# B&R Automation Studio project Doctor
Automation Studio 4.9

## Configuration Doctoring

### Cpu.per - 4PPC70_0702_20B/Cpu.per
```iecst
VAR_CONFIG
	AxisKN AT %M0; (* *)
	AxisRPM AT %M70; (* *)
END_VAR
```

## Configuration WndCLTensCtrl

CPU X20CP1586, AutomationRuntime V4.08, Vc V4.15.4

### Task classes (Cpu.sw)
```
DataObjects: Acp10sys
Binaries: vcctext, arialbd, vcmgr, vccshape, vcnet, Visu03, vcdsloc, vcbclass, vcfntttf, vctcal, vcshared, vcrt, vcpkat, Visu01, vccbmp, vcfile, vccbtn, vcalarm, vccnum, vcpdsw, vcdsint, arial, vccovl, vccline, vcpdvnc, vcctrend, vcgclass, vcpfar00, Visu02, vccpopup, vccddbox, vccbar, sysconf, ashwd, asfw, arconfig, Acp10map, acp10cfg, iomap, vccslider, vccdt, vccstr, TCData
Libraries: AsIecCon, astime, NcGlobal, brsystem, sys_lib, Runtime, powerlnk, fileio, Operator, AsBrMath, dataobj, vcresman
```

### PvMap.vvm - X20CP1586/PvMap.vvm
```iecst
(*Simulation model input parameters*)
VAR_CONFIG
	Cyclic#3.::gControl.Winder.Power AT %Q.::SimModel:SimulationModel.Enable; (*Enable simulation modell if machine is ready*)
	Cyclic#3.::gControl.Line.SetVelocity AT %Q.::SimModel:SetLineVelocity; (*Connect control structure with simulation model*)
	Cyclic#3.::gControl.Winder.SetVelocity AT %Q.::SimModel:SetWinderVelocity; (*Connect control structure with simulation model*)
	Cyclic#3.::gControl.Winder.VelocityCorrection AT %Q.::SimModel:WinderVelocityCorrection; (*Connect control structure with simulation model*)
	Cyclic#3.::gControl.Winder.SetMotorTorque AT %Q.::SimModel:SetMotorTorque; (*Connect control structure with simulation model*)
	Cyclic#3.::gControl.Winder.InitSpeedController AT %Q.::SimModel:InitSpeedController; (*Connect control structure with simulation model*)
	Cyclic#3.::gControl.Winder.ActProportionalGain AT %Q.::SimModel:ActProportionalGain; (*Connect control structure with simulation model*)
	Cyclic#3.::gControl.Winder.ActIntegrationTime AT %Q.::SimModel:ActIntegrationTime; (*Connect control structure with simulation model*)
END_VAR
(*Simulation model output parameters*)
VAR_CONFIG
	::SimModel:SimulationModel.ActLinePosition AT %Q.Cyclic#2.::gControl.Line.ActPosition; (*Connect simulation model with control structure*)
	::SimModel:SimulationModel.ActWinderPosition AT %Q.Cyclic#2.::gControl.Winder.ActPosition; (*Connect simulation model with control structure*)
	::SimModel:SimulationModel.ActMaterialTension AT %Q.Cyclic#2.::gControl.ActMaterialTension; (*Connect simulation model with control structure*)
	::SimModel:SimulationModel.ActLineVelocity AT %Q.Cyclic#2.::gControl.Line.ActVelocity; (*Connect simulation model with control structure*)
	::SimModel:SimulationModel.ActWinderVelocity AT %Q.Cyclic#2.::gControl.Winder.ActVelocity; (*Connect simulation model with control structure*)
	::SimModel:SimulationModel.ActMotorTorque AT %Q.Cyclic#2.::gControl.Winder.ActMotorTorque; (*Connect simulation model with control structure*)
END_VAR
```

## Configuration WndDcrCtrl

### Task classes (Cpu.sw)
```
DataObjects: Acp10sys
Binaries: vcctext, arialbd, vcmgr, vccshape, vcnet, Visu03, vcdsloc, vcbclass, vcfntttf, vctcal, vcshared, vcrt, vcpkat, Visu01, vccbmp, vcfile, vccbtn, vcalarm, vccnum, vcpdsw, vcdsint, arial, vccovl, vccline, vcpdvnc, vcctrend, vcgclass, vcpfar00, Visu02, vccpopup, vccddbox, vccbar, sysconf, ashwd, asfw, iomap, arconfig, Acp10map, acp10cfg, vccslider, vccdt, vccstr, TCData
Libraries: AsIecCon, astime, NcGlobal, brsystem, sys_lib, Runtime, powerlnk, fileio, Operator, AsBrMath, dataobj, vcresman
```

## Logical view

Binary libraries used (declarations not repeated): operator, runtime, astime, AsIecCon, brsystem, sys_lib, AsBrMath, LoopConR, LoopCont, Acp10_MC, Acp10man, Acp10par, NcGlobal, Acp10sim, asstring, standard, vclib, visapi, AsEPL


- Library Logical/Libraries/Library (ANSIC) (no source held here)

### Program Logical/HMI (IEC)

#### Variables.var
```iecst
VAR
	CheckCredentials : BOOL;
	ErrorMessage : STRING[80];
	i : INT;
	Init : BOOL;
	InputPassword : STRING[80]; (*Input taken from HMI*)
	InputUsername : STRING[80]; (*Input taken from HMI*)
	CurrentYear : UINT;
	CurrentSecond : USINT;
	CurrentMonth : USINT;
	CurrentMinute : USINT;
	CurrentHour : USINT;
	CurrentDay : USINT;
	NewYear : UINT;
	NewSecond : USINT;
	NewMonth : USINT;
	NewMinute : USINT;
	NewHour : USINT;
	NewDay : USINT;
	DateTimeSet : UINT; (*Confirms if new date/time was set successfully*)
	SetNewDateTime : BOOL; (*Trigger to apply new date/time*)
	RTC_Get : RTCtime_typ; (*Structure to read current date and time*)
	RTC_Set : RTCtime_typ; (*Structure to set current date and time*)
	Status_RTC : UINT;
	temp_var : BOOL;
END_VAR
```

#### Cyclic.st
```iecst
PROGRAM _CYCLIC
	(* Insert code here *)
	IF(Init = 1)THEN
		Init := 0;
	END_IF

	// Time
	// Reads current date/time from PLC's RTC

	RTC_gettime(ADR(RTC_Get));  // Call PLC's built-in RTC function

	// Update outputs for display
	CurrentYear   := RTC_Get.year;
	CurrentMonth  := RTC_Get.month;
	CurrentDay    := RTC_Get.day;
	CurrentHour   := RTC_Get.hour;
	CurrentMinute := RTC_Get.minute;
	CurrentSecond := RTC_Get.second;

	// Set Date and Time when 'Set Date Time' button is pressed
	IF SetNewDateTime THEN
		IF(temp_var = 0)THEN
			Status_RTC	:= 1;
			temp_var	:= 1;
		END_IF

		RTC_Set.year    := NewYear;
		RTC_Set.month   := NewMonth;
		RTC_Set.day     := NewDay;
		RTC_Set.hour    := NewHour;
		RTC_Set.minute  := NewMinute;
		RTC_Set.second  := NewSecond;

		// Call RTC set function
		Status_RTC := RTC_settime(ADR(RTC_Set));  // Returns TRUE if successful

		IF(Status_RTC = 0)THEN
			SetNewDateTime	:= 0;
			temp_var		:= 0;
		END_IF

	END_IF;

	// Login check
	//	FUNCTION FB_CheckCredentials
	// Credential check
	IF (InputUsername = 'Admin' AND InputPassword = '1234') THEN
		LoginSuccessful := TRUE;
		UserAccessLevel := 1;	// Full access
		CheckCredentials := TRUE;
		ErrorMessage := 'Logged in';
	ELSE
		LoginSuccessful := FALSE;
		UserAccessLevel := 0;	// No input access
		CheckCredentials := FALSE;
		ErrorMessage := 'Wrong user name or password';
	END_IF;

	ErrorMessage := '';   	// Clear any previous message
	InputUsername := '';	// Clear InputUsername field
	InputPassword := '';	// Clear InputPassword field

	IF(Alarm_new = 1)THEN
		Statusdp_alarm	:= 0;
	ELSE
		Statusdp_alarm	:= 1;
	END_IF

END_PROGRAM
```

#### Init.st
```iecst
PROGRAM _INIT
		(*Input of Tension Sensor for 4 axes except main drive *)
	AI1[0]	:= 0;	(*Unwinder Loadcell *)
	AI1[1]	:= 0;	(* Infeed Loadcell *)
	AI1[2]	:= 0;	(* Outfeed Loadcell *)
	AI1[3]	:= 0;	(* Winder Load cell *)
	AI1[4]	:= 0;	(* Dummy Load cell for Main Drive *)

	AI2[0]	:= 0;
	AI2[1]	:= 0;
	AI2[2]	:= 0;
	AI2[3]	:= 0; (*This input is configured for MAIN RPM calculation *)

	(* Input for RPM measurement from drive AI for 4 axes except Winder RPM*)
	AI3[0]	:= 0;   (* Unwinder RPM *)
	AI3[1]	:= 0;	(* Infeed RPM *)
	AI3[2]	:= 0;	(* Outfeed RPM *)
	AI3[3]	:= 0;	(* Winder RPM *)
	AI3[4]	:= 0;	(*This input is configured from AI2[3] for MAIN RPM *)

	AO1[0]	:= 0;
	AO1[1]	:= 0;
	AO1[2]	:= 0;
	AO1[3]	:= 0;

	DI1[0]	:= 0;
	DI1[1]	:= 0;
	DI1[2]	:= 0;
	DI1[3]	:= 0;
	DI1[4]	:= 0;
	DI1[5]	:= 0;
	DI1[6]	:= 0;
	DI1[7]	:= 0;
	DI1[8]	:= 0;
	DI1[9]	:= 0;
	DI1[10]	:= 0;
	DI1[11]	:= 0;

	DI2[0]	:= 0;
	DI2[1]	:= 0;
	DI2[2]	:= 0;
	DI2[3]	:= 0;
	DI2[4]	:= 0;
	DI2[5]	:= 0;
	DI2[6]	:= 0;
	DI2[7]	:= 0;
	DI2[8]	:= 0;
	DI2[9]	:= 0;
	DI2[10]	:= 0;
	DI2[11]	:= 0;

	DO1[0]	:= 0;
	DO1[1]	:= 0;
	DO1[2]	:= 0;
	DO1[3]	:= 0;
	DO1[4]	:= 0;
	DO1[5]	:= 0;
	DO1[6]	:= 0;
	DO1[7]	:= 0;
	DO1[8]	:= 0;
	DO1[9]	:= 0;
	DO1[10]	:= 0;
	DO1[11]	:= 0;

	DO2[0]	:= 0;
	DO2[1]	:= 0;
	DO2[2]	:= 0;
	DO2[3]	:= 0;
	DO2[4]	:= 0;
	DO2[5]	:= 0;
	DO2[6]	:= 0;
	DO2[7]	:= 0;
	DO2[8]	:= 0;
	DO2[9]	:= 0;
	DO2[10]	:= 0;
	DO2[11]	:= 0;

	PageCall	:= 0;
	LastPage	:= 0;
	NewPageReq	:= 0;
	PrevPage	:= 0;
	CurrPage	:= 0;
	DrvComm		:= 0;
	Init		:= 1;
	ParamChange	:= 0;
	NewPage		:= 0;
	SetNewDateTime	:= 0;

END_PROGRAM
```

### Program Logical/Doctoring/HS_Inp_Doct

#### Variables.var
```iecst
VAR
	Encoder_counts : INT;
	ActUnWindKN : LCScINT;
	ActUnWindRPM : LCLiScINT;
	i : USINT;
	Axis_RpmInpFilt : ARRAY[0..4] OF LCPT1;
	HSCounter : LCCounter;
	initialize : BOOL;
	MainRoleDia : INT;
	Axis_KNInpFilt : ARRAY[0..4] OF LCPT1;
	UnwindFilt : LCPT1;
	WindFilt : LCPT1;
	Time_1sec : TON_10ms;
	Old_EncValue : INT;
	Diff_EncValue : INT;
	PulsesPerMin : UDINT;
	UnWindRPM_Scal : LCScINT;
	WindRPM_Scal : LCScINT;
	Numerator : UDINT;
	Denominator : UDINT;
	DriveCurrent_Scal : LCScINT;
	DriveRPM_Scal : LCScINT;
	DriveTorq_Scal : LCScINT;
	DriveFreq_Scal : LCScINT;
END_VAR
```

#### HS_Inp_Init.st
```iecst
PROGRAM _INIT
	(* Insert code here *)
	initialize	:= 1;

	(*Input of Tension Sensor for 4 axes except main drive *)
	AI1[0]	:= 0;	(*Unwinder Loadcell *)
	AI1[1]	:= 0;	(* Infeed Loadcell *)
	AI1[2]	:= 0;	(* Outfeed Loadcell *)
	AI1[3]	:= 0;	(* Winder Load cell *)

	AO1[0]	:= 0;
	AO1[1]	:= 0;
	AO1[2]	:= 0;
	AO1[3]	:= 0;

	DI1[0]	:= 0;
	DI1[1]	:= 0;
	DI1[2]	:= 0;
	DI1[3]	:= 0;
	DI1[4]	:= 0;
	DI1[5]	:= 0;
	DI1[6]	:= 0;
	DI1[7]	:= 0;
	DI1[8]	:= 0;
	DI1[9]	:= 0;
	DI1[10]	:= 0;
	DI1[11]	:= 0;

	DI2[0]	:= 0;
	DI2[1]	:= 0;
	DI2[2]	:= 0;
	DI2[3]	:= 0;
	DI2[4]	:= 0;
	DI2[5]	:= 0;
	DI2[6]	:= 0;
	DI2[7]	:= 0;
	DI2[8]	:= 0;
	DI2[9]	:= 0;
	DI2[10]	:= 0;
	DI2[11]	:= 0;

	DO1[0]	:= 0;
	DO1[1]	:= 0;
	DO1[2]	:= 0;
	DO1[3]	:= 0;
	DO1[4]	:= 0;
	DO1[5]	:= 0;
	DO1[6]	:= 0;
	DO1[7]	:= 0;
	DO1[8]	:= 0;
	DO1[9]	:= 0;
	DO1[10]	:= 0;
	DO1[11]	:= 0;

	DO2[0]	:= 0;
	DO2[1]	:= 0;
	DO2[2]	:= 0;
	DO2[3]	:= 0;
	DO2[4]	:= 0;
	DO2[5]	:= 0;
	DO2[6]	:= 0;
	DO2[7]	:= 0;
	DO2[8]	:= 0;
	DO2[9]	:= 0;
	DO2[10]	:= 0;
	DO2[11]	:= 0;

	i	:= 0;

	IF(Idler.PulsesPerRev = 0)THEN
		Idler.PulsesPerRev	:= 1;
	END_IF

	IF(UnWind.RPM.Actual.Scale.Filter_tim = 0)THEN
		UnWind.RPM.Actual.Scale.Filter_tim	:= 15;
	END_IF

	UnwindFilt.enable	:= 1;
	UnwindFilt.t		:= UnWind.RPM.Actual.Scale.Filter_tim;
	UnwindFilt.basetime	:= HSCounter.mscnt;
	UnwindFilt.set		:= FALSE;
	UnwindFilt.yset		:= 0;

	IF(Wind.RPM.Actual.Scale.Filter_tim = 0)THEN
		Wind.RPM.Actual.Scale.Filter_tim	:= 15;
	END_IF

	WindFilt.enable	:= 1;
	WindFilt.t			:= Wind.RPM.Actual.Scale.Filter_tim;
	WindFilt.basetime	:= HSCounter.mscnt;
	WindFilt.set		:= FALSE;
	WindFilt.yset		:= 0;

	UnWind.Enable	:= 1;
	UnWind.MPM.Enable	:= 1;

	IF((UnWind.RPM.Actual.Scale.InMin = 0)OR(UnWind.RPM.Actual.Scale.InMax = 0))THEN
		UnWind.RPM.Actual.Scale.InMin	:= 1;
		UnWind.RPM.Actual.Scale.InMax	:= 1;
	END_IF

	IF((UnWind.RPM.Actual.Scale.OutMin = 0)OR(UnWind.RPM.Actual.Scale.OutMax = 0))THEN
		UnWind.RPM.Actual.Scale.OutMin	:= 1;
		UnWind.RPM.Actual.Scale.OutMax	:= 1;
	END_IF

	IF((Wind.RPM.Actual.Scale.InMin = 0)OR(Wind.RPM.Actual.Scale.InMax = 0))THEN
		Wind.RPM.Actual.Scale.InMin	:= 1;
		Wind.RPM.Actual.Scale.InMax	:= 1;
	END_IF

	IF((Wind.RPM.Actual.Scale.OutMin = 0)OR(Wind.RPM.Actual.Scale.OutMax = 0))THEN
		Wind.RPM.Actual.Scale.OutMin	:= 1;
		Wind.RPM.Actual.Scale.OutMax	:= 1;
	END_IF

	UnWindRPM_Scal.x1	:= UnWind.RPM.Actual.Scale.InMin;
	UnWindRPM_Scal.x2	:= UnWind.RPM.Actual.Scale.InMax;
	UnWindRPM_Scal.y1	:= UnWind.RPM.Actual.Scale.OutMin;
	UnWindRPM_Scal.y2	:= UnWind.RPM.Actual.Scale.OutMax;

	WindRPM_Scal.x1		:= Wind.RPM.Actual.Scale.InMin;
	WindRPM_Scal.x2		:= Wind.RPM.Actual.Scale.InMax;
	WindRPM_Scal.y1		:= Wind.RPM.Actual.Scale.OutMin;
	WindRPM_Scal.y2		:= Wind.RPM.Actual.Scale.OutMax;

	(* Scaling drive parameters *)
	(* TORQUE *)
	IF((UnWind.Drive.Trq_Scal.InMin = 0)OR(UnWind.Drive.Trq_Scal.InMax = 0))THEN
		UnWind.Drive.Trq_Scal.InMin	:= 1;
		UnWind.Drive.Trq_Scal.InMax	:= 1;
	END_IF

	IF((UnWind.Drive.Trq_Scal.OutMin = 0)OR(UnWind.Drive.Trq_Scal.OutMax = 0))THEN
		UnWind.Drive.Trq_Scal.OutMin 	:= 1;
		UnWind.Drive.Trq_Scal.OutMax := 1;
	END_IF

	IF((Wind.Drive.Trq_Scal.InMin = 0)OR(Wind.Drive.Trq_Scal.InMax = 0))THEN
		Wind.Drive.Trq_Scal.InMin	:= 1;
		Wind.Drive.Trq_Scal.InMax	:= 1;
	END_IF

	IF((Wind.Drive.Trq_Scal.OutMin = 0)OR(Wind.Drive.Trq_Scal.OutMax = 0))THEN
		Wind.Drive.Trq_Scal.OutMin 	:= 1;
		Wind.Drive.Trq_Scal.OutMax := 1;
	END_IF

	(* CURRENT *)
	IF((UnWind.Drive.Current_Scal.InMin = 0)OR(UnWind.Drive.Current_Scal.InMax = 0))THEN
		UnWind.Drive.Current_Scal.InMin	:= 1;
		UnWind.Drive.Current_Scal.InMax	:= 1;
	END_IF

	IF((UnWind.Drive.Current_Scal.OutMin = 0)OR(UnWind.Drive.Current_Scal.OutMax = 0))THEN
		UnWind.Drive.Current_Scal.OutMin 	:= 1;
		UnWind.Drive.Current_Scal.OutMax := 1;
	END_IF

	IF((Wind.Drive.Current_Scal.InMin = 0)OR(Wind.Drive.Current_Scal.InMax = 0))THEN
		Wind.Drive.Current_Scal.InMin	:= 1;
		Wind.Drive.Current_Scal.InMax	:= 1;
	END_IF

	IF((Wind.Drive.Current_Scal.OutMin = 0)OR(Wind.Drive.Current_Scal.OutMax = 0))THEN
		Wind.Drive.Current_Scal.OutMin 	:= 1;
		Wind.Drive.Current_Scal.OutMax := 1;
	END_IF

	(* RPM *)
	IF((UnWind.Drive.RPM_Scal.InMin = 0)OR(UnWind.Drive.RPM_Scal.InMax = 0))THEN
		UnWind.Drive.RPM_Scal.InMin		:= 1;
		UnWind.Drive.RPM_Scal.InMax		:= 1;
	END_IF

	IF((UnWind.Drive.RPM_Scal.OutMin = 0)OR(UnWind.Drive.RPM_Scal.OutMax = 0))THEN
		UnWind.Drive.RPM_Scal.OutMin	:= 1;
		UnWind.Drive.RPM_Scal.OutMax	:= 1;
	END_IF

	IF((Wind.Drive.RPM_Scal.InMin = 0)OR(Wind.Drive.RPM_Scal.InMax = 0))THEN
		Wind.Drive.RPM_Scal.InMin	:= 1;
		Wind.Drive.RPM_Scal.InMax	:= 1;
	END_IF

	(* FREQUENCY *)
	IF((UnWind.Drive.Freq_Scal.InMin = 0)OR(UnWind.Drive.Freq_Scal.InMax = 0))THEN
		UnWind.Drive.Freq_Scal.InMin	:= 1;
		UnWind.Drive.Freq_Scal.InMax	:= 1;
	END_IF

	IF((UnWind.Drive.Freq_Scal.OutMin = 0)OR(UnWind.Drive.Freq_Scal.OutMax = 0))THEN
		UnWind.Drive.Freq_Scal.OutMin 	:= 1;
		UnWind.Drive.Freq_Scal.OutMax := 1;
	END_IF

	IF((Wind.Drive.Freq_Scal.InMin = 0)OR(Wind.Drive.Freq_Scal.InMax = 0))THEN
		Wind.Drive.Freq_Scal.InMin	:= 1;
		Wind.Drive.Freq_Scal.InMax	:= 1;
	END_IF

	IF((Wind.Drive.Freq_Scal.OutMin = 0)OR(Wind.Drive.Freq_Scal.OutMax = 0))THEN
		Wind.Drive.Freq_Scal.OutMin	:= 1;
		Wind.Drive.Freq_Scal.OutMax := 1;
	END_IF

	Time_1sec.PT	:= 100;

(*
	FOR i :=0 TO (MAX_AXES - 1)BY 1 DO
		IF (AxisKN[i].Fact.FilterTime = 0)THEN
			AxisKN[i].Fact.FilterTime	:= 15;
		END_IF

		Axis_KNInpFilt[i].enable		:= TRUE;
		Axis_KNInpFilt[i].t				:= AxisKN[i].Fact.FilterTime;
		Axis_KNInpFilt[i].yset   		:= 0;
		Axis_KNInpFilt[i].basetime 		:= HSCounter.mscnt;
		Axis_KNInpFilt[i].set    		:= FALSE;
	END_FOR;

	FOR i := 0 TO (MAX_AXES - 1) BY 1 DO
		AxisRPM[i].InpBits		:= 0;
		AxisRPM[i].ActRPM		:= 0;

		Axis_RPM[i].x	:= AxisRPM[i].InpBits;
		Axis_RPM[i]();

		AxisKN[i].InpBits		:=	0;
		AxisKN[i].ActTension	:= 0;

		Axis_KN[i].x	:= AxisKN[i].InpBits;
		Axis_KN[i]();
	END_FOR;
*)

	(* UnWinder & Infeed calculation initialization *)

	(*	UnWindFilt.enable	:= 1;
	UnWindFilt.set   	:= 1;
	UnWindFilt.t		:= 0.1;
	UnWindFilt.y_set	:= 0.0;
	UnWindFilt.x 		:= 0.0;
	UnWindFilt();
	UnWindFilt.set   	:= 0;

	ActUnWindKN.x1		:= UnWindKN.MinBits;
	ActUnWindKN.x2		:= UnWindKN.MaxBits;
	ActUnWindKN.y1		:= UnWindKN.MinTension;
	ActUnWindKN.y2		:= UnWindKN.MaxTension;

	InfeedFilt.enable	:= 1;
	InfeedFilt.set   	:= 1;
	InfeedFilt.t		:= 0.1;
	InfeedFilt.y_set	:= 0.0;
	InfeedFilt.x 		:= 0.0;
	InfeedFilt();
	InfeedFilt.set   	:= 0;

	ActInfeedKN.x1		:= InfeedKN.MinBits;
	ActInfeedKN.x2		:= InfeedKN.MaxBits;
	ActInfeedKN.y1		:= InfeedKN.MinTension;
	ActInfeedKN.y2		:= InfeedKN.MaxTension;
*)

	(* Winder & Outfeed calculation initialization *)

(*	WindFilt.enable		:= 1;
	WindFilt.set   		:= 1;
	WindFilt.t			:= 0.1;
	WindFilt.y_set		:= 0.0;
	WindFilt.x 			:= 0.0;
	WindFilt();
	WindFilt.set   		:= 0;

	ActWindKN.x1		:= WinderKN.MinBits;
	ActWindKN.x2		:= WinderKN.MaxBits;
	ActWindKN.y1		:= WinderKN.MinTension;
	ActWindKN.y2		:= WinderKN.MaxTension;

	OutfeedFilt.enable	:= 1;
	OutfeedFilt.set   	:= 1;
	OutfeedFilt.t		:= 0.1;
	OutfeedFilt.y_set	:= 0.0;
	OutfeedFilt.x 		:= 0.0;
	OutfeedFilt();
	OutfeedFilt.set   	:= 0;

	ActOutfeedKN.x1		:= OutfeedKN.MinBits;
	ActOutfeedKN.x2		:= OutfeedKN.MaxBits;
	ActOutfeedKN.y1		:= OutfeedKN.MinTension;
	ActOutfeedKN.y2		:= OutfeedKN.MaxTension;
*)

END_PROGRAM
```

### Program Logical/Doctoring/LS_Inp_OP

#### Variables.var
```iecst
VAR
	check_init : BOOL;
	dec_cnt : USINT;
	inc_cnt : USINT;
	mode_allow : BOOL;
	Mode_Intermediate : BOOL;
	MPMDecTime : TON_10ms;
	MPMIncTime : TON_10ms;
END_VAR
```

#### Cyclic.st
```iecst
PROGRAM _CYCLIC
	(* Insert code here *)
	DigInp.Emergency_OK		:= DI1[0];
	DigInp.Jog_mode			:= DI1[1];
	Mode_Intermediate		:= DI1[2];
	DigInp.MPM_Increase		:= DI1[3];
	DigInp.MPM_Decrease		:= DI1[4];
	DigInp.Safety_Trip		:= DI1[5];

	IF(check_init = 1)THEN
		IF (Mode_Intermediate = 1)THEN
			Alarm_mc[0]	:= 1;
			mode_allow	:= 0;
		ELSE
			mode_allow	:= 1;
		END_IF
		check_init	:= 0;
	END_IF

	IF(mode_allow = 1)THEN
		IF((DigInp.Jog_mode = 0)AND(Mode_Intermediate = 1))THEN
			DigInp.Production_mode	:= Mode_Intermediate;
		ELSE
			DigInp.Production_mode	:= 0;
		END_IF
	ELSE
		DigInp.Production_mode	:= 0;
	END_IF

	IF(DigInp.Production_mode = 1)THEN
		IF(DigInp.MPM_Increase = 1)THEN
			MPMIncTime.IN	:= 1;
			IF(MPMIncTime.ET < 500)THEN
				inc_cnt	:= inc_cnt + 1;
				IF(inc_cnt >= 50)THEN
					UnWind.MPM.SetMPM	:= UnWind.MPM.SetMPM + 1;
					inc_cnt	:= 0;
				END_IF
			ELSIF(MPMIncTime.ET < 800)THEN
				inc_cnt	:= inc_cnt + 1;
				IF(inc_cnt >= 50)THEN
					UnWind.MPM.SetMPM	:= UnWind.MPM.SetMPM + 10;
					inc_cnt	:= 0;
				END_IF
			ELSIF(MPMIncTime.ET < 1000)THEN
				inc_cnt	:= inc_cnt + 1;
				IF(inc_cnt >= 50)THEN
					UnWind.MPM.SetMPM	:= UnWind.MPM.SetMPM + 100;
					inc_cnt	:= 0;
				END_IF
			END_IF
		ELSE
			MPMIncTime.IN	:= 0;
			inc_cnt			:= 0;
		END_IF

		IF(DigInp.MPM_Decrease = 1)THEN
			MPMDecTime.IN	:= 1;
			IF(MPMDecTime.ET < 500)THEN
				dec_cnt	:= dec_cnt + 1;
				IF(dec_cnt >= 50)THEN
					UnWind.MPM.SetMPM	:= UnWind.MPM.SetMPM - 1;
					dec_cnt	:= 0;
				END_IF
			ELSIF(MPMDecTime.ET < 800)THEN
				dec_cnt	:= dec_cnt + 1;
				IF(dec_cnt >= 50)THEN
					UnWind.MPM.SetMPM	:= UnWind.MPM.SetMPM - 10;
					dec_cnt	:= 0;
				END_IF
			ELSIF(MPMDecTime.ET < 1000)THEN
				dec_cnt	:= dec_cnt + 1;
				IF(dec_cnt >= 50)THEN
					UnWind.MPM.SetMPM	:= UnWind.MPM.SetMPM - 100;
					dec_cnt	:= 0;
				END_IF
			END_IF
		ELSE
			MPMDecTime.IN	:= 0;
			dec_cnt			:= 0;
		END_IF
	ELSE
		MPMDecTime.IN	:= 0;
		dec_cnt			:= 0;
		MPMIncTime.IN	:= 0;
		inc_cnt			:= 0;
	END_IF

	IF(DigInp.Production_mode = 1)THEN
		Drive_RW[0].Write_UINT[0]	:= UnWind.MPM.SetMPM;
		Drive_RW[1].Write_UINT[0]	:= DINT_TO_UINT(Drive_RW[0].Read_DINT[2]);
	ELSIF(DigInp.Jog_mode = 1)THEN
		Drive_RW[0].Write_UINT[0]	:= UnWind.MPM.SetMPM;
		Drive_RW[1].Write_UINT[0]	:= Wind.MPM.SetMPM;
	ELSE
		Drive_RW[0].Write_UINT[0]	:= 0;
		Drive_RW[1].Write_UINT[0]	:= 0;
		UnWind.MPM.SetMPM			:= 0;
		Wind.MPM.SetMPM				:= 0;
	END_IF

	MPMIncTime();
	MPMDecTime();

END_PROGRAM
```

- Visualisation Logical/Vis (not shown)

### Program Logical/Alarms (IEC)

#### Variables.var
```iecst
VAR
	i : INT;
	Blink_Trig : TON_10ms;
	count : BOOL;
	Blink_ON : TON_10ms;
	Blink_OFF : TON_10ms;
END_VAR
```

#### Cyclic.st
```iecst
PROGRAM _CYCLIC
	(* Insert code here *)
	Alarm_cnt	:= 0;

	FOR i := 0 TO 99 DO
		IF(Alarms[i] > 0)THEN
			Alarm_cnt	:= Alarm_cnt + 1;
		END_IF
	END_FOR

	IF(Alarm_cnt > 0)THEN
		Statusdp_blink	:= 1;
		IF(count = 0)THEN
			Blink_ON.IN	:= 1;
			IF(Blink_ON.Q = 1)THEN
				count := 1;
				Blink_ON.IN	:= 0;
			END_IF
		ELSE
			Blink_OFF.IN	:= 1;
			IF(Blink_OFF.Q = 1)THEN
				count := 0;
				Blink_OFF.IN := 0;
			END_IF
		END_IF

	ELSE
		Blink_ON.IN		:= 0;
		Blink_OFF.IN	:= 0;
		Statusdp_blink	:= 0;
	END_IF

	Blink_ON(IN := TRUE, PT := 1);	//1 × 10ms = 10 milliseconds
	Blink_OFF(IN := TRUE, PT := 1);

END_PROGRAM
```

#### Init.st
```iecst
PROGRAM _INIT
	(* Insert code here *)
	Statusdp_alarm	:= 0;
	Alarm_cnt		:= 0;
	Alarm_new		:= 0;
	Blink_ON.IN		:= 0;
	Blink_ON.PT		:= 100;
	Blink_OFF.IN	:= 0;
	Blink_OFF.PT	:= 100;

	memset(ADR(Alarms), 0, SIZEOF(Alarms));

END_PROGRAM
```

### Program Logical/EPLCom/EPLCom (IEC)

#### Variables.var
```iecst
VAR
	DataReceived : UINT;
	cnt_enable : BOOL;
	SDO_rd : USINT;
	SDORead1 : EplSDORead;
	DataReceived_INT : INT;
	NMT_Stat : UDINT;
	SDORead2 : EplSDORead;
	Obj_Ident : UDINT;
	tempstat : UINT;
	tempstat_2 : UINT;
END_VAR
VAR CONSTANT
	PLC_INTF : STRING[20] := 'IF1';
END_VAR
VAR
	SDO_rd2 : USINT;
END_VAR
```

#### Cyclic.st
```iecst
PROGRAM _CYCLIC
	(* Insert code here *)

	IF(SDO_rd = 1)THEN
		SDORead1(enable := TRUE);
		IF (SDORead1.status = 0) THEN
//			SDORead1(enable := FALSE);
			SDO_rd	:= SDO_rd + 1;
		ELSIF (SDORead1.status = 20925)THEN
			SDORead1.enable	:= 0;
			tempstat		:= SDORead1.status;
		ELSIF((SDORead1.status >= 31340)AND(SDORead1.status < 65530)) THEN
//			SDORead1(enable := FALSE);
			tempstat	:= SDORead1.status;
		END_IF

	ELSE
//		SDORead1(enable := FALSE);
	END_IF

	IF(SDO_rd2 = 1)THEN
		SDORead2(enable := TRUE);
		IF (SDORead2.status = 0) THEN
//			SDORead2(enable := FALSE);
			SDO_rd2		:= SDO_rd2 + 1;
		ELSIF (SDORead2.status = 20925)THEN
			SDORead2.enable	:= 0;
			tempstat_2		:= SDORead2.status;
		ELSIF ((SDORead2.status >= 31340)AND(SDORead2.status < 65530)) THEN
//			SDORead2(enable := FALSE);
			tempstat_2	:= SDORead2.status;

		END_IF
	ELSE
//		SDORead1(enable := FALSE);
	END_IF

	DataReceived_INT := DataRead_INT;

	IF(cnt_enable = 1)THEN
		DataTobeSent_UINT	:= DataTobeSent_UINT + 1;
	END_IF

END_PROGRAM
```

### Program Logical/EPLCom/EPLCom_Drv1

#### Variables.var
```iecst
VAR
	cnt_enable : BOOL;
	Control_Enable : SINT;
	Control_Enb : USINT;
	Control_WORD : INT;
	DataReceived : UINT;
	DataReceived_INT : INT;
	Derv_Gain : INT;
	dlycnt : USINT := 0;
	dlycnt1 : USINT;
	dlycnt_pid : USINT;
	Drv_Status : INT;
	Ingr_Gain : INT;
	NMT_Stat : UDINT;
	Obj_Ident : UDINT;
	PID_RefSrc : UINT;
	PID_WORD : INT;
END_VAR
VAR CONSTANT
	PLC_INTF : STRING[20] := 'IF1';
END_VAR
VAR
	Porp_Gain : INT;
	rdpid_step : USINT;
	rd_step : USINT;
	RefSrc_WORD : UINT;
	SDORead1 : EplSDORead;
	SDOWrite : EplSDOWrite;
	SDO_pid : BOOL;
	SDO_rd : USINT;
	SDO_rd2 : USINT;
	SDO_wr : USINT;
	Status_WORD : INT;
	step : USINT;
	tempstat : UINT;
	tempstat_2 : UINT;
	wr_step : USINT;
	SDORead_PID : EplSDORead;
	wrpid_step : USINT;
	SDO_pidwr : BOOL;
	dlycnt_wrpid : USINT;
	SDO_PIDWR : EplSDOWrite;
	Prop_Gain : INT;
	DerGain_Set : INT;
	RefSrc_Set : UINT;
	PropGain_Set : INT;
	IntGain_Set : INT;
END_VAR
```

#### Cyclic.st
```iecst
PROGRAM _CYCLIC
	(* Insert code here *)

	CASE rd_step OF
		0:
			IF(SDO_rd = 1)THEN
				rd_step	:= 1;
				dlycnt	:= 0;
			END_IF
		1:
			SDORead1.pData := ADR(Status_WORD); //Data to be read into here
			SDORead1.datalen := 2; //Data length, 2 bytes for 16-bit parameter
			SDORead1.index 		:= 16#200A;
			SDORead1.subindex	:= 40;
			SDORead1.enable		:= 1;
			dlycnt				:= dlycnt + 1;
			IF(dlycnt > 2)THEN
				IF (SDORead1.status = 0) THEN
					SDORead1.enable	:= 0;
					rd_step			:= 2;
					dlycnt			:= 0;
					Drv_Status		:= Status_WORD;
//				ELSIF((SDORead1.status <> 65535)OR(SDORead1.status <> 65534))THEN
				ELSIF(SDORead1.status <> 65535)THEN
					SDORead1.enable	:= 0;
				END_IF
			END_IF

		2:
			SDORead1.pData 		:= ADR(Status_WORD); //Data to be read into here
			SDORead1.datalen 	:= 1; //Data length, 2 bytes for 16-bit parameter
			SDORead1.index 		:= 16#2006;
			SDORead1.subindex	:= 43;
			SDORead1.enable		:= 1;
			dlycnt				:= dlycnt + 1;
			IF(dlycnt > 2)THEN
				IF (SDORead1.status = 0) THEN
					SDORead1.enable	:= 0;
					rd_step			:= 0;
					dlycnt			:= 0;
					SDO_rd			:= 0;
					Control_Enb		:=	INT_TO_USINT(Status_WORD);
//				ELSIF((SDORead1.status <> 65535)OR(SDORead1.status <> 65534))THEN
				ELSIF(SDORead1.status <> 65535)THEN
					SDORead1.enable	:= 0;
				END_IF
			END_IF
	END_CASE

	CASE wr_step OF
		0:
			IF(SDO_wr = 1)THEN
				wr_step	:= 1;
				dlycnt1	:= 0;
			END_IF
		1:

			Control_Enable		:= 0;

			SDOWrite.pData		:= ADR(Control_Enable);
			SDOWrite.datalen 	:= 1; //Data length, 2 bytes for 16-bit parameter
			SDOWrite.index 		:= 16#2006;
			SDOWrite.subindex	:= 43;
			SDOWrite.enable		:= 1;
			dlycnt1				:= dlycnt1 + 1;
			IF(dlycnt1 > 2)THEN
				IF (SDOWrite.status = 0) THEN
					SDOWrite.enable	:= 0;
					wr_step			:= 2;
					dlycnt1			:= 0;
//				ELSIF((SDOWrite.status <> 65535)AND(SDOWrite.status <> 65534))THEN
			ELSIF(SDOWrite.status <> 65535)THEN
					SDOWrite.enable	:= 0;
					SDO_wr			:= 0;
				END_IF
			END_IF

		2:
			Control_WORD		:= 129;

			SDOWrite.pData		:= ADR(Control_WORD);
			SDOWrite.datalen 	:= 2; //Data length, 2 bytes for 16-bit parameter
			SDOWrite.index 		:= 16#2006;
			SDOWrite.subindex	:= 42;
			SDOWrite.enable		:= 1;
			dlycnt1				:= dlycnt1 + 1;
			IF(dlycnt1 > 2)THEN
				IF (SDOWrite.status = 0) THEN
					SDOWrite.enable	:= 0;
					wr_step			:= 0;
					dlycnt1			:= 0;
					SDO_wr			:= 0;
//				ELSIF((SDOWrite.status <> 65535)AND(SDOWrite.status <> 65534))THEN
				ELSIF(SDOWrite.status <> 65535)THEN
					SDOWrite.enable	:= 0;
				END_IF
			END_IF
	END_CASE

	IF(SDO_rd = 0)THEN
		SDORead1.enable	:= 0;
		rd_step			:= 0;
		dlycnt			:= 0;
	END_IF

	IF(SDO_wr = 0)THEN
		SDOWrite.enable	:= 0;
		wr_step			:= 0;
		dlycnt1			:= 0;
	END_IF

	CASE rdpid_step OF
		0:
			IF(SDO_pid = 1)THEN
				rdpid_step	:= 1;
				dlycnt_pid	:= 0;
			END_IF
		1:
			SDORead_PID.pData 		:= ADR(PID_WORD); //Data to be read into here
			SDORead_PID.datalen 	:= 2; //Data length, 2 bytes for 16-bit parameter
			SDORead_PID.index 		:= 16#200E;
			SDORead_PID.subindex	:= 10;
			SDORead_PID.enable		:= 1;
			dlycnt_pid			:= dlycnt_pid + 1;
			IF(dlycnt_pid > 2)THEN
				IF (SDORead_PID.status = 0) THEN
					SDORead_PID.enable	:= 0;
					rdpid_step		:= 2;
					dlycnt_pid		:= 0;
					Porp_Gain		:= PID_WORD;
					//				ELSIF((SDORead_PID.status <> 65535)OR(SDORead_PID.status <> 65534))THEN
				ELSIF(SDORead_PID.status <> 65535)THEN
					SDORead_PID.enable	:= 0;
				END_IF
			END_IF

		2:
			SDORead_PID.pData := ADR(PID_WORD); //Data to be read into here
			SDORead_PID.datalen 	:= 2; //Data length, 2 bytes for 16-bit parameter
			SDORead_PID.index 		:= 16#200E;
			SDORead_PID.subindex	:= 11;
			SDORead_PID.enable		:= 1;
			dlycnt_pid			:= dlycnt_pid + 1;
			IF(dlycnt_pid > 2)THEN
				IF (SDORead_PID.status = 0) THEN
					SDORead_PID.enable	:= 0;
					rdpid_step		:= 3;
					dlycnt_pid		:= 0;
//					SDO_rd			:= 0;
					Ingr_Gain		:= PID_WORD;
//				ELSIF((SDORead_PID.status <> 65535)OR(SDORead_PID.status <> 65534))THEN
				ELSIF(SDORead_PID.status <> 65535)THEN
					SDORead_PID.enable	:= 0;
				END_IF
			END_IF

		3:
			SDORead_PID.pData := ADR(PID_WORD); //Data to be read into here
			SDORead_PID.datalen 	:= 2; //Data length, 2 bytes for 16-bit parameter
			SDORead_PID.index 		:= 16#200E;
			SDORead_PID.subindex	:= 12;
			SDORead_PID.enable		:= 1;
			dlycnt_pid			:= dlycnt_pid + 1;
			IF(dlycnt_pid > 2)THEN
				IF (SDORead_PID.status = 0) THEN
					SDORead_PID.enable	:= 0;
					rdpid_step		:= 4;
					dlycnt_pid		:= 0;
//					SDO_rd			:= 0;
					Derv_Gain		:=	PID_WORD;
//				ELSIF((SDORead_PID.status <> 65535)OR(SDORead_PID.status <> 65534))THEN
				ELSIF(SDORead_PID.status <> 65535)THEN
					SDORead_PID.enable	:= 0;
				END_IF
			END_IF

		4:
			SDORead_PID.pData := ADR(RefSrc_WORD); //Data to be read into here
			SDORead_PID.datalen 	:= 2; //Data length, 2 bytes for 16-bit parameter
			SDORead_PID.index 		:= 16#200E;
			SDORead_PID.subindex	:= 03;
			SDORead_PID.enable		:= 1;
			dlycnt_pid			:= dlycnt_pid + 1;
			IF(dlycnt_pid > 2)THEN
				IF (SDORead_PID.status = 0) THEN
					SDORead_PID.enable	:= 0;
					rdpid_step		:= 0;
					dlycnt_pid		:= 0;
					SDO_pid			:= 0;
					PID_RefSrc		:=	INT_TO_UINT(RefSrc_WORD);
					//				ELSIF((SDORead_PID.status <> 65535)OR(SDORead_PID.status <> 65534))THEN
				ELSIF(SDORead_PID.status <> 65535)THEN
					SDORead_PID.enable	:= 0;
				END_IF
			END_IF
	END_CASE

	CASE wrpid_step OF
		0:
			IF(SDO_pidwr = 1)THEN
				wrpid_step	:= 1;
				dlycnt_wrpid	:= 0;
			END_IF
		1:

			SDO_PIDWR.pData		:= ADR(PropGain_Set);
			SDO_PIDWR.datalen 	:= 2; //Data length, 2 bytes for 16-bit parameter
			SDO_PIDWR.index 	:= 16#200E;
			SDO_PIDWR.subindex	:= 10;
			SDO_PIDWR.enable	:= 1;
			dlycnt_wrpid		:= dlycnt_wrpid + 1;
			IF(dlycnt_wrpid > 2)THEN
				IF (SDO_PIDWR.status = 0) THEN
					SDO_PIDWR.enable	:= 0;
					wrpid_step			:= 2;
					dlycnt_wrpid		:= 0;
					//				ELSIF((SDO_PIDWR.status <> 65535)AND(SDO_PIDWR.status <> 65534))THEN
				ELSIF(SDO_PIDWR.status <> 65535)THEN
					SDO_PIDWR.enable	:= 0;
					SDO_wr				:= 0;
				END_IF
			END_IF

		2:
			SDO_PIDWR.pData		:= ADR(IntGain_Set);
			SDO_PIDWR.datalen 	:= 2; //Data length, 2 bytes for 16-bit parameter
			SDO_PIDWR.index 	:= 16#200E;
			SDO_PIDWR.subindex	:= 11;
			SDO_PIDWR.enable	:= 1;
			dlycnt_wrpid		:= dlycnt_wrpid + 1;
			IF(dlycnt_wrpid > 2)THEN
				IF (SDO_PIDWR.status = 0) THEN
					SDO_PIDWR.enable	:= 0;
					wrpid_step			:= 3;
					dlycnt_wrpid		:= 0;
//				ELSIF((SDO_PIDWR.status <> 65535)AND(SDO_PIDWR.status <> 65534))THEN
				ELSIF(SDO_PIDWR.status <> 65535)THEN
					SDO_PIDWR.enable	:= 0;
				END_IF
			END_IF

		3:
			SDO_PIDWR.pData		:= ADR(DerGain_Set);
			SDO_PIDWR.datalen 	:= 2; //Data length, 2 bytes for 16-bit parameter
			SDO_PIDWR.index 	:= 16#200E;
			SDO_PIDWR.subindex	:= 12;
			SDO_PIDWR.enable	:= 1;
			dlycnt_wrpid		:= dlycnt_wrpid + 1;
			IF(dlycnt_wrpid > 2)THEN
				IF (SDO_PIDWR.status = 0) THEN
					SDO_PIDWR.enable	:= 0;
					wrpid_step			:= 4;
					dlycnt_wrpid		:= 0;
//				ELSIF((SDO_PIDWR.status <> 65535)AND(SDO_PIDWR.status <> 65534))THEN
				ELSIF(SDO_PIDWR.status <> 65535)THEN
					SDO_PIDWR.enable	:= 0;
				END_IF
			END_IF

		4:
			SDO_PIDWR.pData		:= ADR(RefSrc_Set);
			SDO_PIDWR.datalen 	:= 2; //Data length, 2 bytes for 16-bit parameter
			SDO_PIDWR.index 	:= 16#200E;
			SDO_PIDWR.subindex	:= 03;
			SDO_PIDWR.enable	:= 1;
			dlycnt_wrpid		:= dlycnt_wrpid + 1;
			IF(dlycnt_wrpid > 2)THEN
				IF (SDO_PIDWR.status = 0) THEN
					SDO_PIDWR.enable	:= 0;
					wrpid_step			:= 0;
					dlycnt_wrpid		:= 0;
					SDO_wr				:= 0;
					SDO_pidwr			:= 0;
//				ELSIF((SDO_PIDWR.status <> 65535)AND(SDO_PIDWR.status <> 65534))THEN
				ELSIF(SDO_PIDWR.status <> 65535)THEN
					SDO_PIDWR.enable	:= 0;
				END_IF
			END_IF

	END_CASE

	IF(SDO_pid = 0)THEN
		SDORead_PID.enable	:= 0;
		rdpid_step		:= 0;
		dlycnt_pid		:= 0;
	END_IF

	IF(SDO_pidwr = 0)THEN
		SDO_PIDWR.enable	:= 0;
		wrpid_step			:= 0;
		dlycnt_wrpid		:= 0;
	END_IF

	SDORead1();
	SDOWrite();
	SDORead_PID();
	SDO_PIDWR();

	DataReceived_INT := DataRead_INT;

	IF(cnt_enable = 1)THEN
		DataTobeSent_UINT	:= DataTobeSent_UINT + 1;
	END_IF

END_PROGRAM
```

#### Init.st
```iecst
PROGRAM _INIT
	(* Insert code here *)
	(* Get NMT Status *)
	SDORead1.enable	:= 0;
	SDORead1.pDevice := ADR(PLC_INTF); //POWERLINK interface on MN (PLC) ‘IF1’
	SDORead1.node := 3; //Node address is set to 3
	//	SDORead1.index := 16#200A; //Read CAN related parameters starting from 0x1000 - 0x1fff

	SDOWrite.enable		:= 0;
	SDOWrite.node		:= 3;
	SDOWrite.pDevice	:= ADR(PLC_INTF);
	SDOWrite.pData		:= ADR(Control_WORD);
//	SDOWrite.index		:= 16#2006;

	SDORead_PID.enable	:= 0;
	SDORead_PID.pDevice := ADR(PLC_INTF); //POWERLINK interface on MN (PLC) ‘IF1’
	SDORead_PID.node := 3; //Node address is set to 3

	SDO_PIDWR.enable	:= 0;
	SDO_PIDWR.node		:= 3;
	SDO_PIDWR.pDevice	:= ADR(PLC_INTF);
	SDO_PIDWR.pData		:= ADR(Control_WORD);
	//	SDOWrite.index		:= 16#2006;

	DataReceived	:= 25;
	cnt_enable		:= 0;
	SDO_rd			:= 0;

END_PROGRAM
```

### Program Logical/EPLCom/UnWind_Com

#### Variables.var
```iecst
VAR
	cnt_enable : BOOL;
	Control_Enable : SINT;
	Control_Enb : USINT;
	Control_WORD : INT;
	DataReceived : UINT;
	DataReceived_INT : INT;
	DerGain_Set : INT;
	Derv_Gain : INT;
	DIO_Conf : INT;
	dlycnt : USINT := 0;
	dlycnt1 : USINT;
	dlycnt_pid : USINT;
	dlycnt_wrpid : USINT;
	Drv_Status : INT;
	Ingr_Gain : INT;
	init : INT;
	IntGain_Set : INT;
	NMT_Stat : UDINT;
	Obj_Ident : UDINT;
	PID_RefSrc : UINT;
	PID_WORD : INT;
	Porp_Gain : INT;
	PropGain_Set : INT;
	Prop_Gain : INT;
	rdpid_step : USINT;
	rd_step : USINT;
	RefSrc_Set : UINT;
	RefSrc_WORD : UINT;
	SDORead1 : EplSDORead;
	SDORead_PID : EplSDORead;
	SDOWrite : EplSDOWrite;
	SDO_pid : BOOL;
	SDO_pidwr : BOOL;
	SDO_PIDWR : EplSDOWrite;
	SDO_rd : USINT;
	SDO_rd2 : USINT;
	SDO_wr : USINT;
	Status_WORD : INT;
	step : USINT;
	tempstat : UINT;
	tempstat_2 : UINT;
	wrpid_step : USINT;
	wr_step : USINT;
END_VAR
```

#### Cyclic.st
```iecst
PROGRAM _CYCLIC
	(* Insert code here *)

	CASE rd_step OF
		0:
			IF(SDO_rd = 1)THEN
				rd_step	:= 1;
				dlycnt	:= 0;
			END_IF
		1:
			SDORead1.pData := ADR(Status_WORD); //Data to be read into here
			SDORead1.datalen := 2; //Data length, 2 bytes for 16-bit parameter
			SDORead1.index 		:= 16#200A;
			SDORead1.subindex	:= 40;
			SDORead1.enable		:= 1;
			dlycnt				:= dlycnt + 1;
			IF(dlycnt > 2)THEN
				IF (SDORead1.status = 0) THEN
					SDORead1.enable	:= 0;
					rd_step			:= 2;
					dlycnt			:= 0;
					Drv_Status		:= Status_WORD;
//				ELSIF((SDORead1.status <> 65535)OR(SDORead1.status <> 65534))THEN
				ELSIF(SDORead1.status <> 65535)THEN
					SDORead1.enable	:= 0;
				END_IF
			END_IF

		2:
			SDORead1.pData 		:= ADR(Status_WORD); //Data to be read into here
			SDORead1.datalen 	:= 1; //Data length, 2 bytes for 16-bit parameter
			SDORead1.index 		:= 16#2006;
			SDORead1.subindex	:= 43;
			SDORead1.enable		:= 1;
			dlycnt				:= dlycnt + 1;
			IF(dlycnt > 2)THEN
				IF (SDORead1.status = 0) THEN
					SDORead1.enable	:= 0;
					rd_step			:= 0;
					dlycnt			:= 0;
					SDO_rd			:= 0;
					Control_Enb		:=	INT_TO_USINT(Status_WORD);
//				ELSIF((SDORead1.status <> 65535)OR(SDORead1.status <> 65534))THEN
				ELSIF(SDORead1.status <> 65535)THEN
					SDORead1.enable	:= 0;
				END_IF
			END_IF
	END_CASE

	CASE wr_step OF
		0:
			IF((SDO_wr = 1)AND(init = 1))THEN
				wr_step	:= 1;
				dlycnt1	:= 0;
			END_IF
		1:
			Control_Enable		:= 0;

			SDOWrite.pData		:= ADR(Control_Enable);
			SDOWrite.datalen 	:= 1; //Data length, 2 bytes for 16-bit parameter
			SDOWrite.index 		:= 16#2006;
			SDOWrite.subindex	:= 43;
			SDOWrite.enable		:= 1;
			dlycnt1				:= dlycnt1 + 1;
			IF(dlycnt1 > 2)THEN
				IF (SDOWrite.status = 0) THEN
					SDOWrite.enable	:= 0;
					wr_step			:= 2;
					dlycnt1			:= 0;
				ELSIF(SDOWrite.status <> 65535)THEN
					SDOWrite.enable	:= 0;
					SDO_wr			:= 0;
				END_IF
			END_IF

		2:
			Control_WORD		:= 133;

			SDOWrite.pData		:= ADR(Control_WORD);
			SDOWrite.datalen 	:= 2; //Data length, 2 bytes for 16-bit parameter
			SDOWrite.index 		:= 16#2006;
			SDOWrite.subindex	:= 42;
			SDOWrite.enable		:= 1;
			dlycnt1				:= dlycnt1 + 1;
			IF(dlycnt1 > 2)THEN
				IF (SDOWrite.status = 0) THEN
					SDOWrite.enable	:= 0;
					wr_step			:= 3;
					dlycnt1			:= 0;
				ELSIF(SDOWrite.status <> 65535)THEN
					SDOWrite.enable	:= 0;
				END_IF
			END_IF
		3:
			DIO_Conf		:= 0;

			SDOWrite.pData		:= ADR(DIO_Conf);
			SDOWrite.datalen 	:= 2; //Data length, 2 bytes for 16-bit parameter
			SDOWrite.index 		:= 16#2008; //Index = 0x2000 + Menu Number
			SDOWrite.subindex	:= 22;
			SDOWrite.enable		:= 1;
			dlycnt1				:= dlycnt1 + 1;
			IF(dlycnt1 > 2)THEN
				IF (SDOWrite.status = 0) THEN
					SDOWrite.enable	:= 0;
					wr_step			:= 4;
					dlycnt1			:= 0;
					//				ELSIF((SDOWrite.status <> 65535)AND(SDOWrite.status <> 65534))THEN
				ELSIF(SDOWrite.status <> 65535)THEN
					SDOWrite.enable	:= 0;
					SDO_wr			:= 0;
				END_IF
			END_IF

		4:
			DIO_Conf		:= 0;

			SDOWrite.pData		:= ADR(DIO_Conf);
			SDOWrite.datalen 	:= 2; //Data length, 2 bytes for 16-bit parameter
			SDOWrite.index 		:= 16#2008; //Index = 0x2000 + Menu Number
			SDOWrite.subindex	:= 23;
			SDOWrite.enable		:= 1;
			dlycnt1				:= dlycnt1 + 1;
			IF(dlycnt1 > 2)THEN
				IF (SDOWrite.status = 0) THEN
					SDOWrite.enable	:= 0;
					wr_step			:= 5;
					dlycnt1			:= 0;
					//				ELSIF((SDOWrite.status <> 65535)AND(SDOWrite.status <> 65534))THEN
				ELSIF(SDOWrite.status <> 65535)THEN
					SDOWrite.enable	:= 0;
					SDO_wr			:= 0;
				END_IF
			END_IF

		5:
			DIO_Conf		:= 0;

			SDOWrite.pData		:= ADR(DIO_Conf);
			SDOWrite.datalen 	:= 2; //Data length, 2 bytes for 16-bit parameter
			SDOWrite.index 		:= 16#2008; //Index = 0x2000 + Menu Number
			SDOWrite.subindex	:= 24;
			SDOWrite.enable		:= 1;
			dlycnt1				:= dlycnt1 + 1;
			IF(dlycnt1 > 2)THEN
				IF (SDOWrite.status = 0) THEN
					SDOWrite.enable	:= 0;
					wr_step			:= 0;
					dlycnt1			:= 0;
					SDO_wr			:= 0;
					init			:= 0;
				ELSIF(SDOWrite.status <> 65535)THEN
					SDOWrite.enable	:= 0;
					SDO_wr			:= 0;
				END_IF
			END_IF
	END_CASE

	IF((SDO_wr = 1)AND(init = 0))THEN
		//Control_Enable	:= 0;
		SDOWrite.pData		:= ADR(Control_Enable);
		SDOWrite.datalen 	:= 1; //Data length, 2 bytes for 16-bit parameter
		SDOWrite.index 		:= 16#2006;
		SDOWrite.subindex	:= 43;
		SDOWrite.enable		:= 1;
		dlycnt1				:= dlycnt1 + 1;
		IF(dlycnt1 > 2)THEN
			IF (SDOWrite.status = 0) THEN
				SDOWrite.enable	:= 0;
				wr_step			:= 2;
				dlycnt1			:= 0;
			ELSIF(SDOWrite.status <> 65535)THEN
				SDOWrite.enable	:= 0;
				SDO_wr			:= 0;
			END_IF
		END_IF
	END_IF

	IF(SDO_rd = 0)THEN
		SDORead1.enable	:= 0;
		rd_step			:= 0;
		dlycnt			:= 0;
	END_IF

	IF((SDO_wr = 0)AND(init = 0))THEN
		SDOWrite.enable	:= 0;
		wr_step			:= 0;
		dlycnt1			:= 0;
	END_IF

	CASE rdpid_step OF
		0:
			IF(SDO_pid = 1)THEN
				rdpid_step	:= 1;
				dlycnt_pid	:= 0;
			END_IF
		1:
			SDORead_PID.pData 		:= ADR(PID_WORD); //Data to be read into here
			SDORead_PID.datalen 	:= 2; //Data length, 2 bytes for 16-bit parameter
			SDORead_PID.index 		:= 16#200E;
			SDORead_PID.subindex	:= 10;
			SDORead_PID.enable		:= 1;
			dlycnt_pid			:= dlycnt_pid + 1;
			IF(dlycnt_pid > 2)THEN
				IF (SDORead_PID.status = 0) THEN
					SDORead_PID.enable	:= 0;
					rdpid_step		:= 2;
					dlycnt_pid		:= 0;
					Porp_Gain		:= PID_WORD;
					//				ELSIF((SDORead_PID.status <> 65535)OR(SDORead_PID.status <> 65534))THEN
				ELSIF(SDORead_PID.status <> 65535)THEN
					SDORead_PID.enable	:= 0;
				END_IF
			END_IF

		2:
			SDORead_PID.pData := ADR(PID_WORD); //Data to be read into here
			SDORead_PID.datalen 	:= 2; //Data length, 2 bytes for 16-bit parameter
			SDORead_PID.index 		:= 16#200E;
			SDORead_PID.subindex	:= 11;
			SDORead_PID.enable		:= 1;
			dlycnt_pid			:= dlycnt_pid + 1;
			IF(dlycnt_pid > 2)THEN
				IF (SDORead_PID.status = 0) THEN
					SDORead_PID.enable	:= 0;
					rdpid_step		:= 3;
					dlycnt_pid		:= 0;
//					SDO_rd			:= 0;
					Ingr_Gain		:= PID_WORD;
//				ELSIF((SDORead_PID.status <> 65535)OR(SDORead_PID.status <> 65534))THEN
				ELSIF(SDORead_PID.status <> 65535)THEN
					SDORead_PID.enable	:= 0;
				END_IF
			END_IF

		3:
			SDORead_PID.pData := ADR(PID_WORD); //Data to be read into here
			SDORead_PID.datalen 	:= 2; //Data length, 2 bytes for 16-bit parameter
			SDORead_PID.index 		:= 16#200E;
			SDORead_PID.subindex	:= 12;
			SDORead_PID.enable		:= 1;
			dlycnt_pid			:= dlycnt_pid + 1;
			IF(dlycnt_pid > 2)THEN
				IF (SDORead_PID.status = 0) THEN
					SDORead_PID.enable	:= 0;
					rdpid_step		:= 4;
					dlycnt_pid		:= 0;
//					SDO_rd			:= 0;
					Derv_Gain		:=	PID_WORD;
//				ELSIF((SDORead_PID.status <> 65535)OR(SDORead_PID.status <> 65534))THEN
				ELSIF(SDORead_PID.status <> 65535)THEN
					SDORead_PID.enable	:= 0;
				END_IF
			END_IF

		4:
			SDORead_PID.pData := ADR(RefSrc_WORD); //Data to be read into here
			SDORead_PID.datalen 	:= 2; //Data length, 2 bytes for 16-bit parameter
			SDORead_PID.index 		:= 16#200E;
			SDORead_PID.subindex	:= 03;
			SDORead_PID.enable		:= 1;
			dlycnt_pid			:= dlycnt_pid + 1;
			IF(dlycnt_pid > 2)THEN
				IF (SDORead_PID.status = 0) THEN
					SDORead_PID.enable	:= 0;
					rdpid_step		:= 0;
					dlycnt_pid		:= 0;
					SDO_pid			:= 0;
					PID_RefSrc		:=	INT_TO_UINT(RefSrc_WORD);
					//				ELSIF((SDORead_PID.status <> 65535)OR(SDORead_PID.status <> 65534))THEN
				ELSIF(SDORead_PID.status <> 65535)THEN
					SDORead_PID.enable	:= 0;
				END_IF
			END_IF
	END_CASE

	CASE wrpid_step OF
		0:
			IF(SDO_pidwr = 1)THEN
				wrpid_step	:= 1;
				dlycnt_wrpid	:= 0;
			END_IF
		1:

			SDO_PIDWR.pData		:= ADR(PropGain_Set);
			SDO_PIDWR.datalen 	:= 2; //Data length, 2 bytes for 16-bit parameter
			SDO_PIDWR.index 	:= 16#200E;
			SDO_PIDWR.subindex	:= 10;
			SDO_PIDWR.enable	:= 1;
			dlycnt_wrpid		:= dlycnt_wrpid + 1;
			IF(dlycnt_wrpid > 2)THEN
				IF (SDO_PIDWR.status = 0) THEN
					SDO_PIDWR.enable	:= 0;
					wrpid_step			:= 2;
					dlycnt_wrpid		:= 0;
					//				ELSIF((SDO_PIDWR.status <> 65535)AND(SDO_PIDWR.status <> 65534))THEN
				ELSIF(SDO_PIDWR.status <> 65535)THEN
					SDO_PIDWR.enable	:= 0;
					SDO_wr				:= 0;
				END_IF
			END_IF

		2:
			SDO_PIDWR.pData		:= ADR(IntGain_Set);
			SDO_PIDWR.datalen 	:= 2; //Data length, 2 bytes for 16-bit parameter
			SDO_PIDWR.index 	:= 16#200E;
			SDO_PIDWR.subindex	:= 11;
			SDO_PIDWR.enable	:= 1;
			dlycnt_wrpid		:= dlycnt_wrpid + 1;
			IF(dlycnt_wrpid > 2)THEN
				IF (SDO_PIDWR.status = 0) THEN
					SDO_PIDWR.enable	:= 0;
					wrpid_step			:= 3;
					dlycnt_wrpid		:= 0;
//				ELSIF((SDO_PIDWR.status <> 65535)AND(SDO_PIDWR.status <> 65534))THEN
				ELSIF(SDO_PIDWR.status <> 65535)THEN
					SDO_PIDWR.enable	:= 0;
				END_IF
			END_IF

		3:
			SDO_PIDWR.pData		:= ADR(DerGain_Set);
			SDO_PIDWR.datalen 	:= 2; //Data length, 2 bytes for 16-bit parameter
			SDO_PIDWR.index 	:= 16#200E;
			SDO_PIDWR.subindex	:= 12;
			SDO_PIDWR.enable	:= 1;
			dlycnt_wrpid		:= dlycnt_wrpid + 1;
			IF(dlycnt_wrpid > 2)THEN
				IF (SDO_PIDWR.status = 0) THEN
					SDO_PIDWR.enable	:= 0;
					wrpid_step			:= 4;
					dlycnt_wrpid		:= 0;
//				ELSIF((SDO_PIDWR.status <> 65535)AND(SDO_PIDWR.status <> 65534))THEN
				ELSIF(SDO_PIDWR.status <> 65535)THEN
					SDO_PIDWR.enable	:= 0;
				END_IF
			END_IF

		4:
			SDO_PIDWR.pData		:= ADR(RefSrc_Set);
			SDO_PIDWR.datalen 	:= 2; //Data length, 2 bytes for 16-bit parameter
			SDO_PIDWR.index 	:= 16#200E;
			SDO_PIDWR.subindex	:= 03;
			SDO_PIDWR.enable	:= 1;
			dlycnt_wrpid		:= dlycnt_wrpid + 1;
			IF(dlycnt_wrpid > 2)THEN
				IF (SDO_PIDWR.status = 0) THEN
					SDO_PIDWR.enable	:= 0;
					wrpid_step			:= 0;
					dlycnt_wrpid		:= 0;
					SDO_wr				:= 0;
					SDO_pidwr			:= 0;
//				ELSIF((SDO_PIDWR.status <> 65535)AND(SDO_PIDWR.status <> 65534))THEN
				ELSIF(SDO_PIDWR.status <> 65535)THEN
					SDO_PIDWR.enable	:= 0;
				END_IF
			END_IF

	END_CASE

	IF(SDO_pid = 0)THEN
		SDORead_PID.enable	:= 0;
		rdpid_step			:= 0;
		dlycnt_pid			:= 0;
	END_IF

	IF(SDO_pidwr = 0)THEN
		SDO_PIDWR.enable	:= 0;
		wrpid_step			:= 0;
		dlycnt_wrpid		:= 0;
	END_IF

	SDORead1();
	SDOWrite();
	SDORead_PID();
	SDO_PIDWR();

	DataReceived_INT := DataRead_INT;

	IF(cnt_enable = 1)THEN
		DataTobeSent_UINT	:= DataTobeSent_UINT + 1;
	END_IF

END_PROGRAM
```

#### Init.st
```iecst
PROGRAM _INIT
	(* Insert code here *)
	(* Get NMT Status *)
	SDORead1.enable	:= 0;
	SDORead1.pDevice := ADR(PLC_INTF); //POWERLINK interface on MN (PLC) ‘IF1’
	SDORead1.node := 3; //Node address is set to 3
	//	SDORead1.index := 16#200A; //Read CAN related parameters starting from 0x1000 - 0x1fff

	SDOWrite.enable		:= 0;
	SDOWrite.node		:= 3;
	SDOWrite.pDevice	:= ADR(PLC_INTF);
	SDOWrite.pData		:= ADR(Control_WORD);
//	SDOWrite.index		:= 16#2006;

	SDORead_PID.enable	:= 0;
	SDORead_PID.pDevice := ADR(PLC_INTF); //POWERLINK interface on MN (PLC) ‘IF1’
	SDORead_PID.node := 3; //Node address is set to 3

	SDO_PIDWR.enable	:= 0;
	SDO_PIDWR.node		:= 3;
	SDO_PIDWR.pDevice	:= ADR(PLC_INTF);
	SDO_PIDWR.pData		:= ADR(Control_WORD);
	//	SDOWrite.index		:= 16#2006;

	DataReceived	:= 25;
	cnt_enable		:= 0;
	SDO_rd			:= 0;
	init			:= 1;
	SDO_wr			:= 1;
END_PROGRAM
```

### Program Logical/EPLCom/Wind_Com

#### Variables.var
```iecst
VAR
	cnt_enable : BOOL := 00;
	Control_Enable : INT;
	Control_Enb : USINT := 0;
	Control_WORD : INT;
	DataReceived : UINT;
	DataReceived_INT : INT := 0;
	DerGain_Set : INT;
	Derv_Gain : INT;
	DIO_Conf : INT := 0;
	dlycnt : USINT := 0;
	dlycnt1 : USINT := 0;
	dlycnt_pid : USINT := 0;
	dlycnt_wrpid : USINT;
	Drv_Status : INT := 0;
	Ingr_Gain : INT;
	init : INT;
	IntGain_Set : INT;
	PID_RefSrc : UINT;
	PID_WORD : INT;
	Porp_Gain : INT;
	PropGain_Set : INT;
	Prop_Gain : INT;
	rdpid_step : USINT := 0;
	rd_step : USINT;
	RefSrc_Set : UINT;
	RefSrc_WORD : UINT;
	SDORead1 : EplSDORead;
	SDORead_PID : EplSDORead;
	SDOWrite : EplSDOWrite;
	SDO_pid : BOOL := FALSE;
	SDO_pidwr : BOOL;
	SDO_PIDWR : EplSDOWrite;
	SDO_rd : BOOL := FALSE;
	SDO_wr : USINT := 0;
	Status_WORD : INT := 0;
	wrpid_step : USINT;
	wr_step : USINT := 0;
END_VAR
```

#### Cyclic.st
```iecst
PROGRAM _CYCLIC
	(* Insert code here *)

	CASE rd_step OF
		0:
			IF(SDO_rd = 1)THEN
				rd_step	:= 1;
				dlycnt	:= 0;
			END_IF
		1:
			SDORead1.pData := ADR(Status_WORD); //Data to be read into here
			SDORead1.datalen := 2; //Data length, 2 bytes for 16-bit parameter
			SDORead1.index 		:= 16#200A;
			SDORead1.subindex	:= 40;
			SDORead1.enable		:= 1;
			dlycnt				:= dlycnt + 1;
			IF(dlycnt > 2)THEN
				IF (SDORead1.status = 0) THEN
					SDORead1.enable	:= 0;
					rd_step			:= 2;
					dlycnt			:= 0;
					Drv_Status		:= Status_WORD;
				ELSIF(SDORead1.status <> 65535)THEN
					SDORead1.enable	:= 0;
				END_IF
			END_IF

		2:
			SDORead1.pData 		:= ADR(Status_WORD); //Data to be read into here
			SDORead1.datalen 	:= 1; //Data length, 2 bytes for 16-bit parameter
			SDORead1.index 		:= 16#2006;
			SDORead1.subindex	:= 43;
			SDORead1.enable		:= 1;
			dlycnt				:= dlycnt + 1;
			IF(dlycnt > 2)THEN
				IF (SDORead1.status = 0) THEN
					SDORead1.enable	:= 0;
					rd_step			:= 0;
					dlycnt			:= 0;
					SDO_rd			:= 0;
					Control_Enb		:=	INT_TO_USINT(Status_WORD);
				ELSIF(SDORead1.status <> 65535)THEN
					SDORead1.enable	:= 0;
				END_IF
			END_IF
	END_CASE

	CASE wr_step OF
		0:
			IF((SDO_wr = 1)AND(init = 1))THEN
				wr_step	:= 1;
				dlycnt1	:= 0;
			END_IF
		1:
			Control_Enable		:= 0;

			SDOWrite.pData		:= ADR(Control_Enable);
			SDOWrite.datalen 	:= 1; //Data length, 2 bytes for 16-bit parameter
			SDOWrite.index 		:= 16#2006;
			SDOWrite.subindex	:= 43;
			SDOWrite.enable		:= 1;
			dlycnt1				:= dlycnt1 + 1;
			IF(dlycnt1 > 2)THEN
				IF (SDOWrite.status = 0) THEN
					SDOWrite.enable	:= 0;
					wr_step			:= 2;
					dlycnt1			:= 0;
				ELSIF(SDOWrite.status <> 65535)THEN
					SDOWrite.enable	:= 0;
					SDO_wr			:= 0;
				END_IF
			END_IF

		2:
			Control_WORD		:= 133;

			SDOWrite.pData		:= ADR(Control_WORD);
			SDOWrite.datalen 	:= 2; //Data length, 2 bytes for 16-bit parameter
			SDOWrite.index 		:= 16#2006;
			SDOWrite.subindex	:= 42;
			SDOWrite.enable		:= 1;
			dlycnt1				:= dlycnt1 + 1;
			IF(dlycnt1 > 2)THEN
				IF (SDOWrite.status = 0) THEN
					SDOWrite.enable	:= 0;
					wr_step			:= 3;
					dlycnt1			:= 0;
				ELSIF(SDOWrite.status <> 65535)THEN
					SDOWrite.enable	:= 0;
				END_IF
			END_IF
		3:
			DIO_Conf		:= 0;

			SDOWrite.pData		:= ADR(DIO_Conf);
			SDOWrite.datalen 	:= 2; //Data length, 2 bytes for 16-bit parameter
			SDOWrite.index 		:= 16#2008; //Index = 0x2000 + Menu Number
			SDOWrite.subindex	:= 22;
			SDOWrite.enable		:= 1;
			dlycnt1				:= dlycnt1 + 1;
			IF(dlycnt1 > 2)THEN
				IF (SDOWrite.status = 0) THEN
					SDOWrite.enable	:= 0;
					wr_step			:= 4;
					dlycnt1			:= 0;
					//				ELSIF((SDOWrite.status <> 65535)AND(SDOWrite.status <> 65534))THEN
				ELSIF(SDOWrite.status <> 65535)THEN
					SDOWrite.enable	:= 0;
					SDO_wr			:= 0;
				END_IF
			END_IF

		4:
			DIO_Conf		:= 0;

			SDOWrite.pData		:= ADR(DIO_Conf);
			SDOWrite.datalen 	:= 2; //Data length, 2 bytes for 16-bit parameter
			SDOWrite.index 		:= 16#2008; //Index = 0x2000 + Menu Number
			SDOWrite.subindex	:= 23;
			SDOWrite.enable		:= 1;
			dlycnt1				:= dlycnt1 + 1;
			IF(dlycnt1 > 2)THEN
				IF (SDOWrite.status = 0) THEN
					SDOWrite.enable	:= 0;
					wr_step			:= 5;
					dlycnt1			:= 0;
					//				ELSIF((SDOWrite.status <> 65535)AND(SDOWrite.status <> 65534))THEN
				ELSIF(SDOWrite.status <> 65535)THEN
					SDOWrite.enable	:= 0;
					SDO_wr			:= 0;
				END_IF
			END_IF

		5:
			DIO_Conf		:= 0;

			SDOWrite.pData		:= ADR(DIO_Conf);
			SDOWrite.datalen 	:= 2; //Data length, 2 bytes for 16-bit parameter
			SDOWrite.index 		:= 16#2008; //Index = 0x2000 + Menu Number
			SDOWrite.subindex	:= 24;
			SDOWrite.enable		:= 1;
			dlycnt1				:= dlycnt1 + 1;
			IF(dlycnt1 > 2)THEN
				IF (SDOWrite.status = 0) THEN
					SDOWrite.enable	:= 0;
					wr_step			:= 0;
					dlycnt1			:= 0;
					SDO_wr			:= 0;
					init			:= 0;
				ELSIF(SDOWrite.status <> 65535)THEN
					SDOWrite.enable	:= 0;
					SDO_wr			:= 0;
				END_IF
			END_IF
	END_CASE

	IF((SDO_wr = 1)AND(init = 0))THEN
		//Control_Enable	:= 0;
		SDOWrite.pData		:= ADR(Control_Enable);
		SDOWrite.datalen 	:= 1; //Data length, 2 bytes for 16-bit parameter
		SDOWrite.index 		:= 16#2006;
		SDOWrite.subindex	:= 43;
		SDOWrite.enable		:= 1;
		dlycnt1				:= dlycnt1 + 1;
		IF(dlycnt1 > 2)THEN
			IF (SDOWrite.status = 0) THEN
				SDOWrite.enable	:= 0;
				wr_step			:= 2;
				dlycnt1			:= 0;
			ELSIF(SDOWrite.status <> 65535)THEN
				SDOWrite.enable	:= 0;
				SDO_wr			:= 0;
			END_IF
		END_IF
	END_IF

	IF(SDO_rd = 0)THEN
		SDORead1.enable	:= 0;
		rd_step			:= 0;
		dlycnt			:= 0;
	END_IF

	IF((SDO_wr = 0) AND (init = 0))THEN
		SDOWrite.enable	:= 0;
		wr_step			:= 0;
		dlycnt1			:= 0;
	END_IF

	CASE rdpid_step OF
		0:
			IF(SDO_pid = 1)THEN
				rdpid_step	:= 1;
				dlycnt_pid	:= 0;
			END_IF
		1:
			SDORead_PID.pData 		:= ADR(PID_WORD); //Data to be read into here
			SDORead_PID.datalen 	:= 2; //Data length, 2 bytes for 16-bit parameter
			SDORead_PID.index 		:= 16#200E;
			SDORead_PID.subindex	:= 10;
			SDORead_PID.enable		:= 1;
			dlycnt_pid			:= dlycnt_pid + 1;
			IF(dlycnt_pid > 2)THEN
				IF (SDORead_PID.status = 0) THEN
					SDORead_PID.enable	:= 0;
					rdpid_step		:= 2;
					dlycnt_pid		:= 0;
					Prop_Gain		:= PID_WORD;
				ELSIF(SDORead_PID.status <> 65535)THEN
					SDORead_PID.enable	:= 0;
				END_IF
			END_IF

		2:
			SDORead_PID.pData := ADR(PID_WORD); //Data to be read into here
			SDORead_PID.datalen 	:= 2; //Data length, 2 bytes for 16-bit parameter
			SDORead_PID.index 		:= 16#200E;
			SDORead_PID.subindex	:= 11;
			SDORead_PID.enable		:= 1;
			dlycnt_pid			:= dlycnt_pid + 1;
			IF(dlycnt_pid > 2)THEN
				IF (SDORead_PID.status = 0) THEN
					SDORead_PID.enable	:= 0;
					rdpid_step		:= 3;
					dlycnt_pid		:= 0;
					Ingr_Gain		:= PID_WORD;
				ELSIF(SDORead_PID.status <> 65535)THEN
					SDORead_PID.enable	:= 0;
				END_IF
			END_IF

		3:
			SDORead_PID.pData := ADR(PID_WORD); //Data to be read into here
			SDORead_PID.datalen 	:= 2; //Data length, 2 bytes for 16-bit parameter
			SDORead_PID.index 		:= 16#200E;
			SDORead_PID.subindex	:= 12;
			SDORead_PID.enable		:= 1;
			dlycnt_pid			:= dlycnt_pid + 1;
			IF(dlycnt_pid > 2)THEN
				IF (SDORead_PID.status = 0) THEN
					SDORead_PID.enable	:= 0;
					rdpid_step		:= 4;
					dlycnt_pid		:= 0;
					Derv_Gain		:=	PID_WORD;
				ELSIF(SDORead_PID.status <> 65535)THEN
					SDORead_PID.enable	:= 0;
				END_IF
			END_IF

		4:
			SDORead_PID.pData := ADR(RefSrc_WORD); //Data to be read into here
			SDORead_PID.datalen 	:= 2; //Data length, 2 bytes for 16-bit parameter
			SDORead_PID.index 		:= 16#200E;
			SDORead_PID.subindex	:= 03;
			SDORead_PID.enable		:= 1;
			dlycnt_pid			:= dlycnt_pid + 1;
			IF(dlycnt_pid > 2)THEN
				IF (SDORead_PID.status = 0) THEN
					SDORead_PID.enable	:= 0;
					rdpid_step		:= 0;
					dlycnt_pid		:= 0;
					SDO_pid			:= 0;
					PID_RefSrc		:=	INT_TO_UINT(RefSrc_WORD);
				ELSIF(SDORead_PID.status <> 65535)THEN
					SDORead_PID.enable	:= 0;
				END_IF
			END_IF
	END_CASE

	CASE wrpid_step OF
		0:
			IF(SDO_pidwr = 1)THEN
				wrpid_step	:= 1;
				dlycnt_wrpid	:= 0;
			END_IF
		1:

			SDO_PIDWR.pData		:= ADR(PropGain_Set);
			SDO_PIDWR.datalen 	:= 2; //Data length, 2 bytes for 16-bit parameter
			SDO_PIDWR.index 	:= 16#200E;
			SDO_PIDWR.subindex	:= 10;
			SDO_PIDWR.enable	:= 1;
			dlycnt_wrpid		:= dlycnt_wrpid + 1;
			IF(dlycnt_wrpid > 2)THEN
				IF (SDO_PIDWR.status = 0) THEN
					SDO_PIDWR.enable	:= 0;
					wrpid_step			:= 2;
					dlycnt_wrpid		:= 0;
					//				ELSIF((SDO_PIDWR.status <> 65535)AND(SDO_PIDWR.status <> 65534))THEN
				ELSIF(SDO_PIDWR.status <> 65535)THEN
					SDO_PIDWR.enable	:= 0;
					SDO_wr				:= 0;
				END_IF
			END_IF

		2:
			SDO_PIDWR.pData		:= ADR(IntGain_Set);
			SDO_PIDWR.datalen 	:= 2; //Data length, 2 bytes for 16-bit parameter
			SDO_PIDWR.index 	:= 16#200E;
			SDO_PIDWR.subindex	:= 11;
			SDO_PIDWR.enable	:= 1;
			dlycnt_wrpid		:= dlycnt_wrpid + 1;
			IF(dlycnt_wrpid > 2)THEN
				IF (SDO_PIDWR.status = 0) THEN
					SDO_PIDWR.enable	:= 0;
					wrpid_step			:= 3;
					dlycnt_wrpid		:= 0;
					//				ELSIF((SDO_PIDWR.status <> 65535)AND(SDO_PIDWR.status <> 65534))THEN
				ELSIF(SDO_PIDWR.status <> 65535)THEN
					SDO_PIDWR.enable	:= 0;
				END_IF
			END_IF

		3:
			SDO_PIDWR.pData		:= ADR(DerGain_Set);
			SDO_PIDWR.datalen 	:= 2; //Data length, 2 bytes for 16-bit parameter
			SDO_PIDWR.index 	:= 16#200E;
			SDO_PIDWR.subindex	:= 12;
			SDO_PIDWR.enable	:= 1;
			dlycnt_wrpid		:= dlycnt_wrpid + 1;
			IF(dlycnt_wrpid > 2)THEN
				IF (SDO_PIDWR.status = 0) THEN
					SDO_PIDWR.enable	:= 0;
					wrpid_step			:= 4;
					dlycnt_wrpid		:= 0;
					//				ELSIF((SDO_PIDWR.status <> 65535)AND(SDO_PIDWR.status <> 65534))THEN
				ELSIF(SDO_PIDWR.status <> 65535)THEN
					SDO_PIDWR.enable	:= 0;
				END_IF
			END_IF

		4:
			SDO_PIDWR.pData		:= ADR(RefSrc_Set);
			SDO_PIDWR.datalen 	:= 2; //Data length, 2 bytes for 16-bit parameter
			SDO_PIDWR.index 	:= 16#200E;
			SDO_PIDWR.subindex	:= 03;
			SDO_PIDWR.enable	:= 1;
			dlycnt_wrpid		:= dlycnt_wrpid + 1;
			IF(dlycnt_wrpid > 2)THEN
				IF (SDO_PIDWR.status = 0) THEN
					SDO_PIDWR.enable	:= 0;
					wrpid_step			:= 0;
					dlycnt_wrpid		:= 0;
					SDO_wr				:= 0;
					SDO_pidwr			:= 0;
					//				ELSIF((SDO_PIDWR.status <> 65535)AND(SDO_PIDWR.status <> 65534))THEN
				ELSIF(SDO_PIDWR.status <> 65535)THEN
					SDO_PIDWR.enable	:= 0;
				END_IF
			END_IF

	END_CASE

	IF(SDO_pid = 0)THEN
		SDORead_PID.enable	:= 0;
		rdpid_step			:= 0;
		dlycnt_pid			:= 0;
	END_IF

	IF(SDO_pidwr = 0)THEN
		SDO_PIDWR.enable	:= 0;
		wrpid_step			:= 0;
		dlycnt_wrpid		:= 0;
	END_IF

	SDORead1();
	SDOWrite();
	SDORead_PID();
	SDO_PIDWR();

	DataReceived_INT := DataRead_INT;

	IF(cnt_enable = 1)THEN
		DataTobeSent_UINT	:= DataTobeSent_UINT + 1;
	END_IF

END_PROGRAM
```

#### Init.st
```iecst
PROGRAM _INIT
	(* Insert code here *)
	(* Insert code here *)
	(* Get NMT Status *)
	SDORead1.enable	:= 0;
	SDORead1.pDevice := ADR(PLC_INTF); //POWERLINK interface on MN (PLC) ‘IF1’
	SDORead1.node := 4; //Node address is set to 3
	//	SDORead1.index := 16#200A; //Read CAN related parameters starting from 0x1000 - 0x1fff

	SDOWrite.enable		:= 0;
	SDOWrite.node		:= 4;
	SDOWrite.pDevice	:= ADR(PLC_INTF);
	SDOWrite.pData		:= ADR(Control_WORD);
	//	SDOWrite.index		:= 16#2006;

	SDORead_PID.enable	:= 0;
	SDORead_PID.pDevice := ADR(PLC_INTF); //POWERLINK interface on MN (PLC) ‘IF1’
	SDORead_PID.node := 4; //Node address is set to 3

	SDO_PIDWR.enable	:= 0;
	SDO_PIDWR.node		:= 4;
	SDO_PIDWR.pDevice	:= ADR(PLC_INTF);
	SDO_PIDWR.pData		:= ADR(Control_WORD);
	//	SDOWrite.index		:= 16#2006;

	DataReceived	:= 25;
	cnt_enable		:= 0;
	SDO_rd			:= 0;
	init			:= 1;
	SDO_wr			:= 1;
END_PROGRAM
```

Listed in the project but not available here: Logical/Global.typ, Logical/Global.var, Logical/UnWindTC, Logical/5Drive
